FUNCTION_BLOCK FB_07
VAR_INPUT
	TRONG AT %I* : BOOL;
END_VAR
VAR_OUTPUT
END_VAR
VAR
END_VAR

END_FUNCTION_BLOCK

(* stored: Version 1.1.0.1, ProductVersion 3.1.4024.12
   POU FB_07: Id {f0f54cd0-3d63-4265-b0b7-3a5a4db3a3a7}, SpecialFunc None *)
